PROGRAM Debounce
VAR
	Input: BOOL;
	TON_0: TON;
	TOF_0: TOF;
	DelayOn: BOOL;
	DelayOff: BOOL;
	DebouncedInput: BOOL;
END_VAR

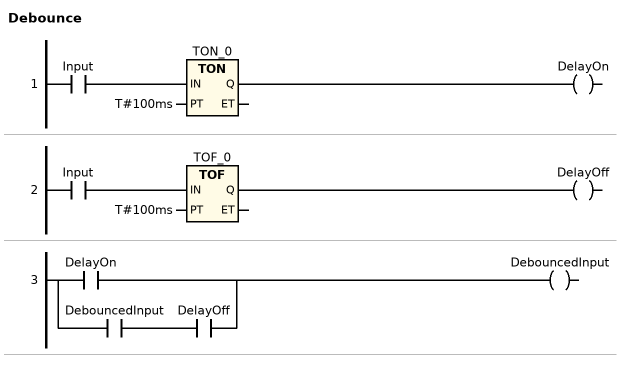
// NETWORK 1
TON_0(IN := Input, PT := T#100ms); // TON
DelayOn := TON_0.Q;

// NETWORK 2
TOF_0(IN := Input, PT := T#100ms); // TOF
DelayOff := TOF_0.Q;

// NETWORK 3
DebouncedInput := DelayOn OR DebouncedInput AND DelayOff;

END_PROGRAM

(* stored: Version 1.1.0.1, ProductVersion 3.1.4024.10
   POU Debounce: Id {6fd6a7d6-41c1-430f-916c-6e29cfc5862d}, SpecialFunc None *)
